// TIA Portal project "babu_conveyor" (V15)

(* hardware
DEVICE "S7-1200 station_1"  S7-1200 Station
   slot 0: "Rack_0"  S7-1200 Rack  Rack  V1.0
   slot 1: "PLC_1"  CPU 1212C DC/DC/DC  6ES7 212-1AE40-0XB0  V4.2
*)

// ===== PLC "PLC_1"  CPU 1212C DC/DC/DC =====

VAR_GLOBAL   // PLC tag table "Default tag table"
   "SWITCH" AT %M0.0 : Bool;
   "BOTTLE SENSOR" AT %M0.1 : Bool;
   "LIGHT" AT %Q0.2 : Bool;
   "CONVEYOR" AT %Q0.3 : Bool;
   "FILL BOTTLE" AT %Q0.4 : Bool;
   "MEMORY" AT %M0.5 : Bool;
END_VAR

// folder: System blocks/Program resources

DATA_BLOCK "IEC_Timer_0_DB_1"   // DB2
{ S7_Optimized_Access := 'TRUE' }
AUTHOR : Simatic
FAMILY : IEC
NAME : IEC_TMR
VERSION : 1.0
// stored: InstanceOfName IEC_TIMER
"IEC_TIMER"
BEGIN
END_DATA_BLOCK

// folder: (top level)

ORGANIZATION_BLOCK "Main"   // OB1, LAD, ProgramCycle
TITLE = "Main Program Sweep (Cycle)"
{ S7_Optimized_Access := 'TRUE' }
VERSION : 0.1
   VAR_INPUT
      Initial_Call : Bool;   // Initial call of this OB
      Remanence : Bool;   // =True, if remanent data are available
   END_VAR
BEGIN

REGION Network 1
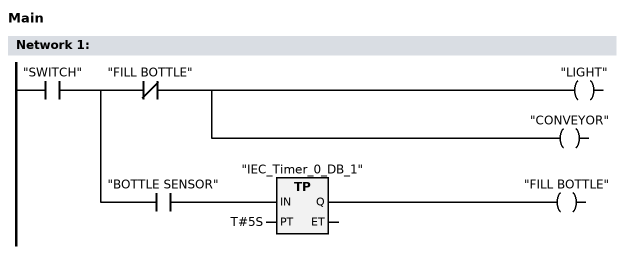
   "LIGHT" := "SWITCH" AND NOT "FILL BOTTLE";
   "CONVEYOR" := "LIGHT";
   "IEC_Timer_0_DB_1".TP(IN := "SWITCH" AND "BOTTLE SENSOR", PT := T#5S);
   "FILL BOTTLE" := "IEC_Timer_0_DB_1".Q;
END_REGION
END_ORGANIZATION_BLOCK